PROGRAM MAIN
VAR
	stStructure : ST_SampleValue;
	bFlag : BOOL := FALSE;
	nNum : DINT := 0;
END_VAR

IF NOT bFlag THEN

bFlag := TRUE;
END_IF
F_UpdateValue(stStructure);
F_UpdateUsingVAR(nNUM);

END_PROGRAM

(* stored: Version 1.1.0.1, ProductVersion 3.1.4024.16
   POU MAIN: Id {9b5f34b6-2067-4d5e-9e23-748a9ef51e2b}, SpecialFunc None *)
